// TIA Portal V17 export
// export: Created 2025-05-22T06:01:10.1102621Z, ExportSetting WithDefaults, DisplayName Totally Integrated Automation Portal, DisplayVersion V17 Update 8, DisplayName TIA Portal Openness, DisplayVersion V17 Update 8, DisplayName TIA Portal Version Control Interface, DisplayVersion V17, DisplayName SINAMICS Startdrive Advanced, DisplayVersion V17 SP2, DisplayName SINAMICS Startdrive G110M, G120, G120C, G120D, G120P, G115D, DisplayVersion V17 SP2, DisplayName SINAMICS Startdrive G130, G150, S120, S150, SINAMICS MV, S210, DisplayVersion V17 SP2, DisplayName STEP 7 Professional, DisplayVersion V17 Update 8, DisplayName SINUMERIK ONE STEP 7 Toolbox, DisplayVersion V17 Update 12, DisplayName SINUMERIK ONE PLC Basic Program Plus, DisplayVersion V17 Update 12, DisplayName SINUMERIK 840D sl STEP 7 Toolbox, DisplayVersion V17 Update 12, DisplayName STEP 7 Safety, DisplayVersion V17 Update 6, DisplayName WinCC Advanced, DisplayVersion V17 Update 8
DATA_BLOCK "DB6801_UNIT_2_DOWN_SEALING_STRUCTURE"   // DB6801
AUTHOR : ETXETAR
VERSION : 1.0
// stored: AutoNumber false, DBAccessibleFromOPCUA true, DBAccessibleFromWebserver true, InstanceOfName FB6502_SEALING_STRUCTURES, InstanceOfType FB
"FB6502_SEALING_STRUCTURES"
   // VAR_INPUT
   //    OPTIONS_0 : Byte;
   //    CLOSED_1_I : Bool;
   //    CLOSED_2_I : Bool;
   //    CLOSED_3_I : Bool;
   //    CLOSED_4_I : Bool;
   //    OPENED_1_I : Bool;
   //    OPENED_2_I : Bool;
   //    OPENED_3_I : Bool;
   //    OPENED_4_I : Bool;
   //    CLOSE_CONDITIONS : Bool;
   //    OPEN_CONDITIONS : Bool;
   //    HMI_LINE_REQUEST : Bool;
   //    CLOSE_AUTO_REQUEST : Bool;
   //    OPEN_AUTO_REQUEST_1 : Bool;
   //    UNIT_ALARM : UInt;
   //    STATION_ALARM : UInt;
   // END_VAR
   // VAR_OUTPUT
   //    CLOSED : Bool;
   //    OPENED : Bool;
   //    CLOSED_1_ALARM : Bool;
   //    CLOSED_2_ALARM : Bool;
   //    CLOSED_3_ALARM : Bool;
   //    CLOSED_4_ALARM : Bool;
   //    OPENED_1_ALARM : Bool;
   //    OPENED_2_ALARM : Bool;
   //    OPENED_3_ALARM : Bool;
   //    OPENED_4_ALARM : Bool;
   //    HMI_MOTION_EXECUTABILITY_LEFT : Bool;
   //    HMI_MOTION_EXECUTABILITY_RIGHT : Bool;
   //    HMI_MOTION_END_POS_LEFT : Bool;
   //    HMI_MOTION_END_POS_RIGHT : Bool;
   //    HMI_MOTION_ACTIVE_LEFT : Bool;
   //    HMI_MOTION_ACTIVE_RIGHT : Bool;
   //    CLOSE : Bool;
   //    OPEN : Bool;
   // END_VAR
   // VAR
   //    CYL { S7_SetPoint := 'True'} : "OPEN_CLOSE_HATCH_CLADDING";
   //    TIMER_CLOSED { S7_SetPoint := 'True'} : TON_TIME;
   //    TIMER_OPENED { S7_SetPoint := 'True'} : TON_TIME;
   //    TIMER_SIMULTANEITY { S7_SetPoint := 'True'} : TON_TIME;
   //    TIMER_TIME_EXCEEDED { S7_SetPoint := 'True'} : TON_TIME;
   // END_VAR
BEGIN
END_DATA_BLOCK
